// TIA Portal V17 export
// export: Created 2022-07-20T06:59:49.7547926Z, ExportSetting WithDefaults, DisplayName Totally Integrated Automation Portal, DisplayVersion V17, DisplayName TIA Portal Openness, DisplayVersion V17, DisplayName TIA Portal Version Control Interface, DisplayVersion V17, DisplayName SINAMICS Startdrive Advanced, DisplayVersion V17, DisplayName SINAMICS Startdrive G130, G150, S120, S150, SINAMICS MV, S210, DisplayVersion V17, DisplayName SINAMICS Startdrive G110M, G120, G120C, G120D, G120P, G115D, DisplayVersion V17, DisplayName STEP 7 Professional, DisplayVersion V17, DisplayName STEP 7 Safety, DisplayVersion V17, DisplayName WinCC Advanced, DisplayVersion V17
FUNCTION_BLOCK "FB10020_MovingAverage"   // FB10020, LAD
{ S7_Optimized_Access := 'TRUE' }
VERSION : 0.1
// stored: AutoNumber false, IsIECCheckEnabled false, IsRetainMemResEnabled false, MemoryReserve 100, SetENOAutomatically false, UDAEnableTagReadback false
   VAR_INPUT
      Entry : LReal;
   END_VAR
   VAR_OUTPUT
      MovingAverage : LReal;
   END_VAR
   VAR_IN_OUT
      NumberOfMovingValues : Int;   // From 1 to 50
   END_VAR
   VAR
      i : Int;
      NumberOfValidEntryValues : Int;
      SumMovingValues : LReal;
      R_TRIG_Clock_2Hz : R_TRIG;
      R_TRIG_DeleteOldValues { S7_SetPoint := 'True'} : R_TRIG;
      Values : Array[0..50] of LReal;
   END_VAR
BEGIN

REGION Network 1 (SCL): First Scan
   IF
       "FirstScan"
   THEN
       FOR #i := 0 TO 50 DO
           #Values[#i] := 1.0e308;
       END_FOR;
   END_IF;
END_REGION

REGION Network 2 (SCL): Edge Signals & Timers
   REGION EDGE SIGNALS
       #R_TRIG_Clock_2Hz(CLK := "Clock_2Hz");
       #R_TRIG_DeleteOldValues(CLK := #NumberOfValidEntryValues > #NumberOfMovingValues);
   END_REGION

   REGION TIMERS
   END_REGION
END_REGION

REGION Network 3 (SCL): Moving Average CommandsManagement
   REGION BOUNDARIES
       IF
           #NumberOfMovingValues < 1
       THEN
           #NumberOfMovingValues := 1;
       ELSIF
           #NumberOfMovingValues > 50
       THEN
           #NumberOfMovingValues := 50;
       END_IF;
   END_REGION
END_REGION

REGION Network 4 (SCL): Moving Average Management
   //Determine How Many Values On The Array Are Valid
   FOR #i := 0 TO 50 DO
       IF
           #Values[#i] = 1.0e308
       THEN
           #NumberOfValidEntryValues := #i;
           EXIT;
       END_IF;
   END_FOR;

   //Record Entry Values
   IF
       #R_TRIG_Clock_2Hz.Q
   THEN
       FOR #i := 0 TO 50 DO
           IF
               #Values[#i] <> 1.0e308
           THEN
               #Values[#i] := #Entry;
               EXIT;
           END_IF;
       END_FOR;
   END_IF;

   //Delete Old Entry Values
   IF
       #R_TRIG_DeleteOldValues.Q
   THEN
       FOR #i := 1 TO 50 DO
           #Values[#i - 1] := #Values[#i];
       END_FOR;
   END_IF;

   //Calculate Moving Average Value
   "FC10024_ArrayAverage"("Array" := #Values,
                          NumberOfValues := #NumberOfValidEntryValues,
                          Average => #MovingAverage);
END_REGION
END_FUNCTION_BLOCK
